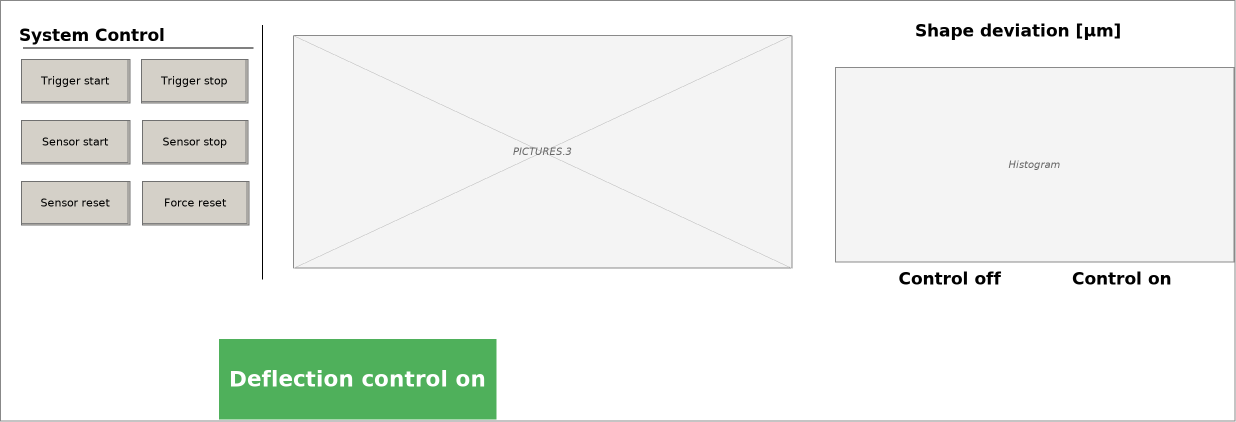
VISUALIZATION VISUALISATION_DEFLEC_CONTROL  // 1236x422
    Button (21,59 109x44), "Trigger start"
        OnMouseClick: execute { VARIABLES.CAN_TRIGGER_STATE:=1; }
    Button (141,59 107x44), "Trigger stop"
        OnMouseClick: execute { VARIABLES.CAN_TRIGGER_STATE:=0; }
    Button (21,120 109x44), "Sensor start"
        OnMouseClick: execute { CAN_CONTROL_STATE:=1; }
    Button (142,120 106x44), "Sensor stop"
        OnMouseClick: execute { CAN_CONTROL_STATE:=0; }
    Button (21,181 109x44), "Sensor reset"
        OnMouseClick: execute { CAN_CONTROL_STATE:=2; }
    Button (142,181 107x44), "Force reset"
        OnMouseClick: execute { VARIABLES.FORCE_RESET:=1; }
    Rectangle (17,20 150x30), "System Control"
    Line (253,48) (23,48)
    Rectangle (1056,265 132x27), "Control on"
    Rectangle (871,265 158x27), "Control off"
    Line (262,25) (262,279)
    Rectangle (896,17 245x27), "Shape deviation [µm]"
    Image (293,35 499x233), image: PICTURES.3
    Histogram (835,67 399x195), scale format: %.1f, scale 0..60
        p1518820177: VARIABLES.RESULT
        p102497268: VARIABLES.RESULT
        p788070771: ARRAY [0..1] OF REAL
    Rectangle (218,338 279x82), "Deflection control on", invisible if: DEFLECTION_CONTROL_ON<>1
END_VISUALIZATION

(* stored: Version 1.1.0.1, ProductVersion 3.1.0.26
   Visu VISUALISATION_DEFLEC_CONTROL: Id {be525aa1-56e5-4c74-9e33-5d4eb3b052b1} *)
